FUNCTION_BLOCK Motor (* Basic Function Block Type *)
  (* Standard: 61499-2 *)
  (* Version 0.0, 2011-12-21, 4DIAC-IDE, 4DIAC-Consortium *)
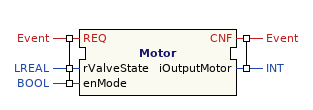
  EVENT_INPUT
    REQ WITH rValveState, enMode; (* Normal Execution Request *)
  END_EVENT
  EVENT_OUTPUT
    CNF WITH iOutputMotor; (* Execution Confirmation *)
  END_EVENT
  VAR_INPUT
    rValveState : LREAL; (* Input event qualifier *)
    enMode : BOOL;
  END_VAR
  VAR_OUTPUT
    iOutputMotor : INT; (* Output event qualifier *)
  END_VAR
  VAR
    iMotor : INT; (* Internal Variable *)
    rValveStateBefore : LREAL := 0; (* Internal Variable *)
    counter : INT := 0; (* Internal Variable *)
  END_VAR
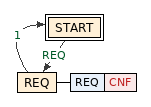
  EC_STATES
    START; (* Initial State *)
    REQ : REQ -> CNF; (* Normal execution *)
  END_STATES
  EC_TRANSITIONS
    START TO REQ := REQ;
    REQ TO START := 1;
  END_TRANSITIONS
  ALGORITHM REQ IN ST: (* Normally executed algorithm *)
IF (enMode=0) THEN
		(*iOutputMotor := CIEC_INT ( rValveState,0.0, (rMaxFeedwaterPressure * rMaxValveState),0, 10000);*)
	iOutputMotor := CIEC_INT(rValveState);
	ELSE
		IF ( (counter MOD 25) = 0) THEN
			iMotor:= CIEC_INT((rValveState - rValveStateBefore)*1000);
			rValveStateBefore :=rValveState;
		END_IF
		counter := counter+1;
		iOutputMotor := iMotor;
END_IF
  END_ALGORITHM
END_FUNCTION_BLOCK
